// TwinCAT 3 PLC project Plc
// Title: inxton
// Company: Inxton
// ProjectVersion: 0.0.0.0
// ProgramVersion: 3.1.4023.0
// libraries:
//   Tc2_Standard, * (Beckhoff Automation GmbH)
//   Tc2_System, * (Beckhoff Automation GmbH)
//   Tc3_Module, * (Beckhoff Automation GmbH)
// project tree:
//   / PlcTask.TcTTO
//   POUs/ MAIN.TcPOU, Data.TcDUT, Math.TcDUT
// real-time tasks:
//   TASK PlcTask: cycle T#11ms, priority 20, ADS port 350

CONFIGURATION Plc
    RESOURCE PLC ON TwinCAT3
        TASK PlcTask(INTERVAL := T#11ms, PRIORITY := 20);
        PROGRAM MAIN WITH PlcTask : MAIN;
    END_RESOURCE
END_CONFIGURATION

// ---- POUs/Data.TcDUT
TYPE
    Data :
    STRUCT
        IncrementDouble : REAL;
		IncrementInt : INT;
		
		DoubleValue:REAL;
		IntValue : INT;
		Recipe : STRING;
    END_STRUCT
END_TYPE

// ---- POUs/Math.TcDUT
TYPE
    Math :
    STRUCT
        Sinus : LREAL;
		NegativeSinus : LREAL;
		
		Cosinus : LREAL;
		Tangent : LREAL;
    END_STRUCT
END_TYPE

// ---- POUs/MAIN.TcPOU
PROGRAM MAIN
VAR
	Data :Data;
	Math : Math;
END_VAR

Data.IncrementDouble := 0.005;
Data.IncrementInt := 1;
Data.DoubleValue := Data.DoubleValue + Data.IncrementDouble ;
if Data.DoubleValue >= 3.141592653 then
//	Data.DoubleValue := 0;
end_if; 
Data.IntValue := ABS(LREAL_TO_INT(Data.DoubleValue*100)) MOD 1000;
 
Math.Sinus := SIN(Data.DoubleValue);
Math.NegativeSinus := SIN(-Data.DoubleValue);
Math.Cosinus := COS(Data.DoubleValue);
Math.Tangent := TAN(Data.DoubleValue);

END_PROGRAM
